INTERFACE ITF_Sensor_TestDecorator EXTENDS ITF_Sensor

METHOD PUBLIC SetContact
VAR_INPUT
	bIN: BOOL;
END_VAR
END_METHOD

END_INTERFACE

(* stored: Version 1.1.0.1
   Itf ITF_Sensor_TestDecorator: Id {a0f2d16b-b657-44ae-a8cc-b4101f3dfa25}
   Method SetContact: Id {8f48095d-bf4c-4e86-8462-502e949f6b96} *)
